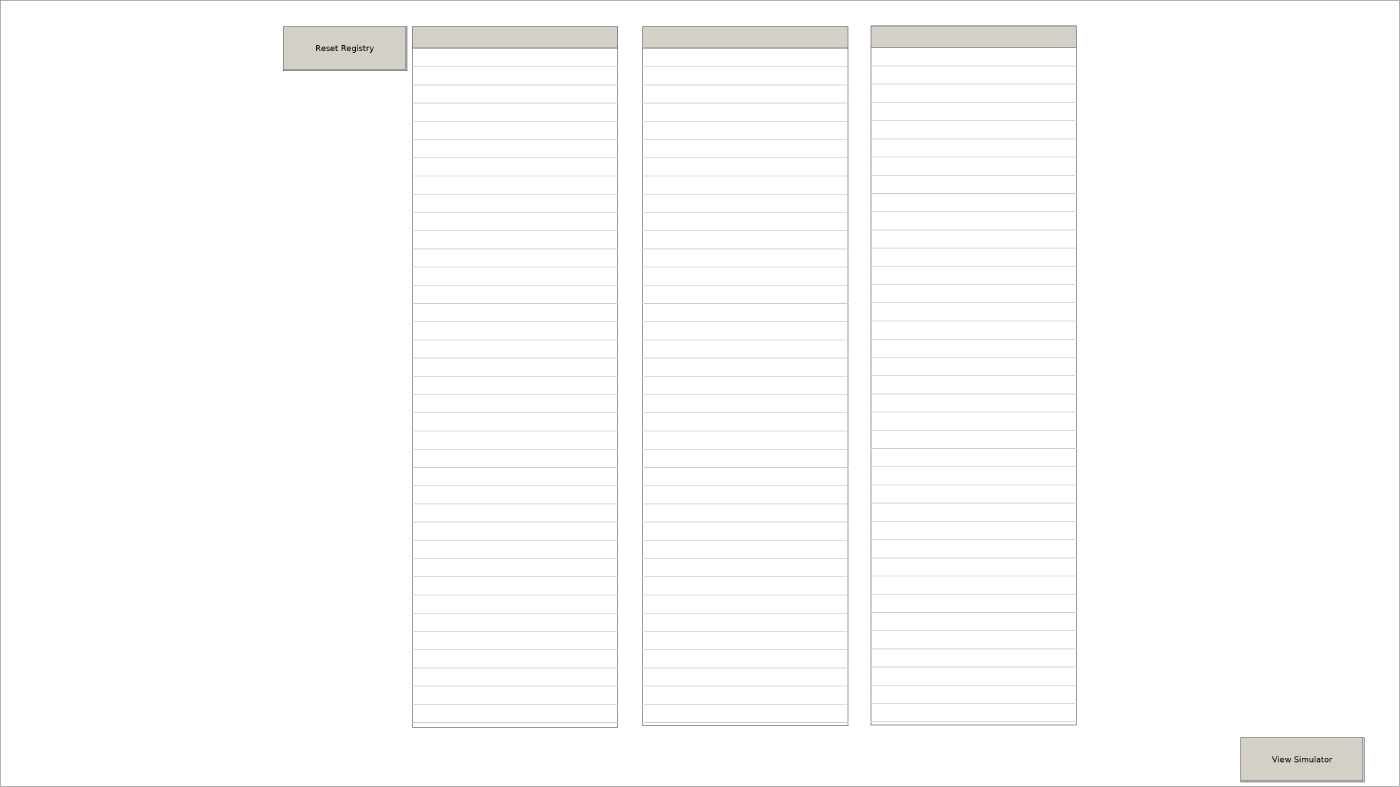
VISUALIZATION TimeStampOnItems  // 1920x1080
    Table (565,36 282x962), data array: PRG_ReadTime.aDigitalSensorTime
        p3854506369: PRG_ReadTime.aDigitalSensorTime[INDEX]
        p2232123230: Digital Sensor Timestamp
    Table (881,36 282x960), data array: PRG_ReadTime.aTCPPortCameraTime
        p3854506369: PRG_ReadTime.aTCPPortCameraTime[INDEX]
        p2232123230: TCP Camera Timestamp
    Button (388,36 170x61), "Reset Registry"
        OnMouseDown: execute { GVL_HMI.stTimestampCmd.bResetRegistry := TRUE; }
    Button (1701,1012 170x61), "View Simulator"
        OnMouseClick: change screen: ItemSimulator
    Table (1194,35 282x960), data array: PRG_ReadTime.aDeltaTimeMS
        p3854506369: PRG_ReadTime.aDeltaTimeMS[INDEX]
        p2232123230: Delta Time in MS
END_VISUALIZATION

(* stored: Version 1.1.0.1, ProductVersion 3.1.4024.12
   Visu TimeStampOnItems: Id {f2d56eba-13d1-4ae5-8e51-aa1a021d4f87} *)
